// TIA Portal V20 export
DATA_BLOCK "Instance_FB_Digita_Inputs_DB"   // DB101
// stored: AutoNumber false, InstanceOfName FB_Digita_Inputs, InstanceOfType FB
"FB_Digita_Inputs"
   // VAR_INPUT
   //    "I-Digital_Input_0" : Bool;
   //    "I-Digital_Input_1" : Bool;
   //    "I-Digital_Input_2" : Bool;
   //    "I-Digital_Input_3" : Bool;
   //    "I-Digital_Input_4" : Bool;
   //    "I-Digital_Input_5" : Bool;
   //    "I-Digital_Input_6" : Bool;
   //    "I-Digital_Input_7" : Bool;
   //    "I-Digital_Input_8" : Bool;
   //    "I-Digital_Input_9" : Bool;
   //    "I-Digital_Input_10" : Bool;
   //    "I-Digital_Input_11" : Bool;
   //    "I-Digital_Input_12" : Bool;
   //    "I-Digital_Input_13" : Bool;
   // END_VAR
   // VAR_OUTPUT
   //    DB_Digital_Input_0 : Bool;
   //    DB_Digital_Input_1 : Bool;
   //    DB_Digital_Input_2 : Bool;
   //    DB_Digital_Input_3 : Bool;
   //    DB_Digital_Input_4 : Bool;
   //    DB_Digital_Input_5 : Bool;
   //    DB_Digital_Input_6 : Bool;
   //    DB_Digital_Input_7 : Bool;
   //    DB_Digital_Input_8 : Bool;
   //    DB_Digital_Input_9 : Bool;
   //    DB_Digital_Input_10 : Bool;
   //    DB_Digital_Input_11 : Bool;
   //    DB_Digital_Input_12 : Bool;
   //    DB_Digital_Input_13 : Bool;
   // END_VAR
BEGIN
END_DATA_BLOCK
